(* Logix 5000 project; controller Sucrose_Main Emulate 5570 rev 20.12; software revision 20.01; part 15 of 30 *)
(* tags used below, declared in another part *)
   Alarm_ACK_Master_Timer : TIMER;
   DI_E22_0 : ALIAS FOR FLX_E22:0:I;   // Discrete Input EN2T_FLX 192.168.1.22
   DO_E22_2 : ALIAS FOR FLX_E22:2:O;   // Discrete Output EN2T_FLX 192.168.1.22
   DO_E22_3 : ALIAS FOR FLX_E22:3:O;   // Discrete Output EN2T_FLX 192.168.1.22
   DO_E22_4 : ALIAS FOR FLX_E22:4:O;   // Discrete Output EN2T_FLX 192.168.1.22
   FV140501_AOI : QSI_Flow_Valve;   // FV-14-05-01 PRE FILTER TRAIN 1 SUPPLY VALVE
   FV140502_AOI : QSI_Flow_Valve;   // FV-14-05-02 FINAL FILTER TRAIN 1 SUPPLY VALVE
   FV140503_AOI : QSI_Flow_Valve;   // FV-14-05-03 HOT WATER LOW POINT DRAIN VALVE
   FV140601_AOI : QSI_Flow_Valve;   // FV-14-06-01 PRE FILTER TRAIN 2 SUPPLY VALVE
   FV140602_AOI : QSI_Flow_Valve;   // FV-14-06-02 FINAL FILTER TRAIN 2 SUPPLY VALVE
   FV150501_AOI : QSI_Flow_Valve;   // FV-15-05-01 DIVERT TO SCRAP OR TO DRAIN VALVE
   FV230500_AOI : QSI_Flow_Valve;   // FV-23-05-00 SUCROSE LOW POINT DRAIN VALVE
   FV230601_AOI : QSI_Flow_Valve;   // FV-23-06-01-O PRE FILTER TRAIN 2 INLET VALVE OPEN
   FV230606_AOI : QSI_Flow_Valve;   // FV-23-06-06-O PRE FILTER TRAIN 2 OUTLET VALVE OPEN
   FV230608_AOI : QSI_Flow_Valve;   // FV-23-06-08-O FINAL FILTER TRAIN 2 INLET VALVE OPEN
   FV230613_AOI : QSI_Flow_Valve;   // FV-23-06-13-O FINAL FILTER TRAIN 2 OUTLET VALVE OPEN
   Sucrose_MM_Enable : BOOL;
   SucroseCIP_FILTRATION_REMOTE : CIP_REMOTE;
   SucroseFiltration : Area_Program;
(* FiltrationArea_EN2T_IO_Discrete_DO_E22_2, continued *)

ROUTINE _12_FV230601   (* ladder *)
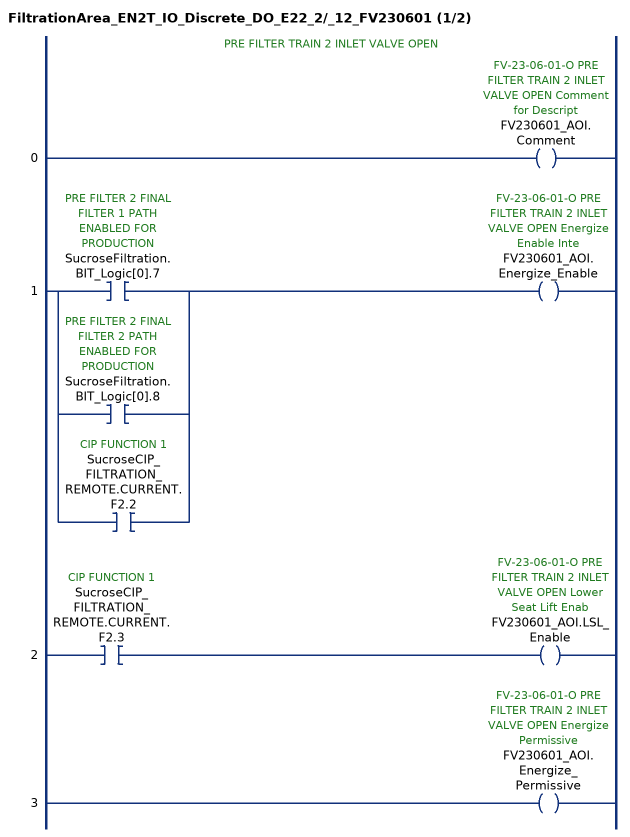
   // PRE FILTER TRAIN 2 INLET VALVE OPEN
   0: OTE(FV230601_AOI.Comment);
   1: [XIC(SucroseFiltration.BIT_Logic[0].7) ,XIC(SucroseFiltration.BIT_Logic[0].8) ,XIC(SucroseCIP_FILTRATION_REMOTE.CURRENT.F2.2) ]OTE(FV230601_AOI.Energize_Enable);
   2: XIC(SucroseCIP_FILTRATION_REMOTE.CURRENT.F2.3)OTE(FV230601_AOI.LSL_Enable);
   3: OTE(FV230601_AOI.Energize_Permissive);
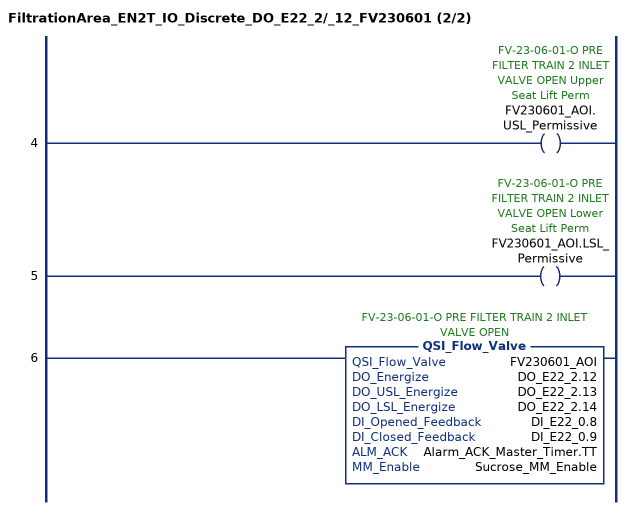
   4: OTE(FV230601_AOI.USL_Permissive);
   5: OTE(FV230601_AOI.LSL_Permissive);
   6: QSI_Flow_Valve(FV230601_AOI,DO_E22_2.12,DO_E22_2.13,DO_E22_2.14,DI_E22_0.8,DI_E22_0.9,Alarm_ACK_Master_Timer.TT,Sucrose_MM_Enable);
END_ROUTINE

ROUTINE MainRoutine   (* ladder *)
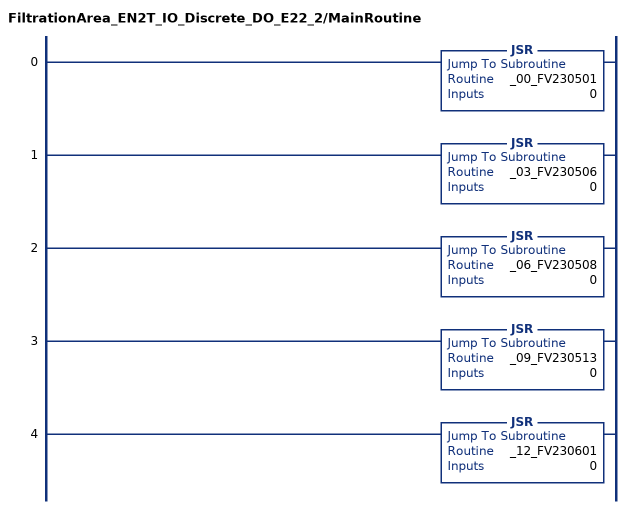
   0: JSR(_00_FV230501,0);
   1: JSR(_03_FV230506,0);
   2: JSR(_06_FV230508,0);
   3: JSR(_09_FV230513,0);
   4: JSR(_12_FV230601,0);
END_ROUTINE
END_PROGRAM

PROGRAM FiltrationArea_EN2T_IO_Discrete_DO_E22_3   (* main routine MainRoutine *)

ROUTINE _00_FV230606   (* ladder *)
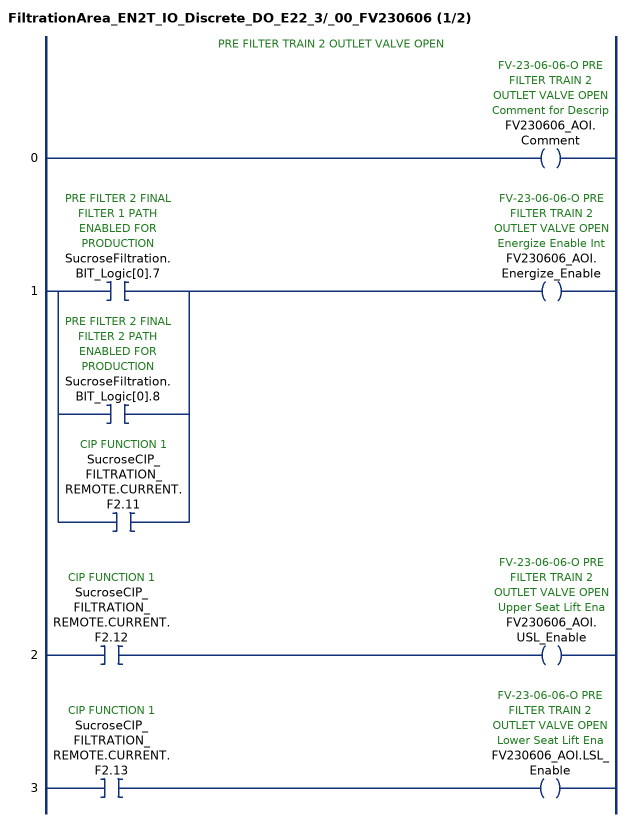
   // PRE FILTER TRAIN 2 OUTLET VALVE OPEN
   0: OTE(FV230606_AOI.Comment);
   1: [XIC(SucroseFiltration.BIT_Logic[0].7) ,XIC(SucroseFiltration.BIT_Logic[0].8) ,XIC(SucroseCIP_FILTRATION_REMOTE.CURRENT.F2.11) ]OTE(FV230606_AOI.Energize_Enable);
   2: XIC(SucroseCIP_FILTRATION_REMOTE.CURRENT.F2.12)OTE(FV230606_AOI.USL_Enable);
   3: XIC(SucroseCIP_FILTRATION_REMOTE.CURRENT.F2.13)OTE(FV230606_AOI.LSL_Enable);
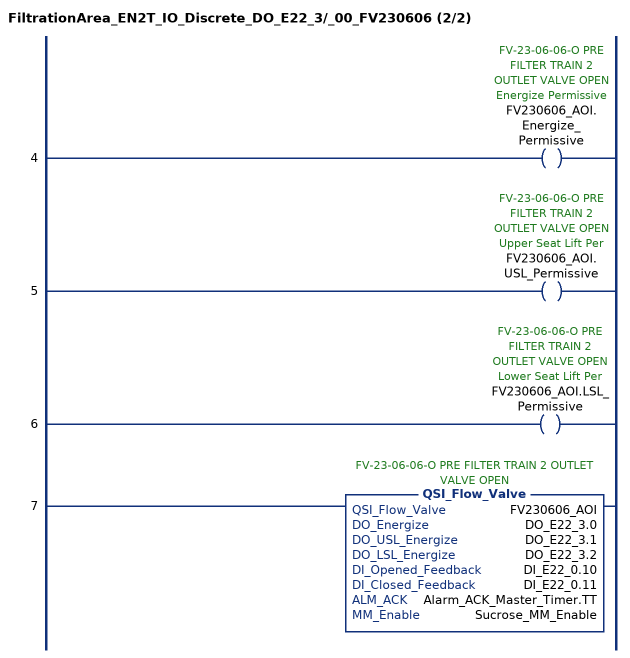
   4: OTE(FV230606_AOI.Energize_Permissive);
   5: OTE(FV230606_AOI.USL_Permissive);
   6: OTE(FV230606_AOI.LSL_Permissive);
   7: QSI_Flow_Valve(FV230606_AOI,DO_E22_3.0,DO_E22_3.1,DO_E22_3.2,DI_E22_0.10,DI_E22_0.11,Alarm_ACK_Master_Timer.TT,Sucrose_MM_Enable);
END_ROUTINE

ROUTINE _03_FV230608   (* ladder *)
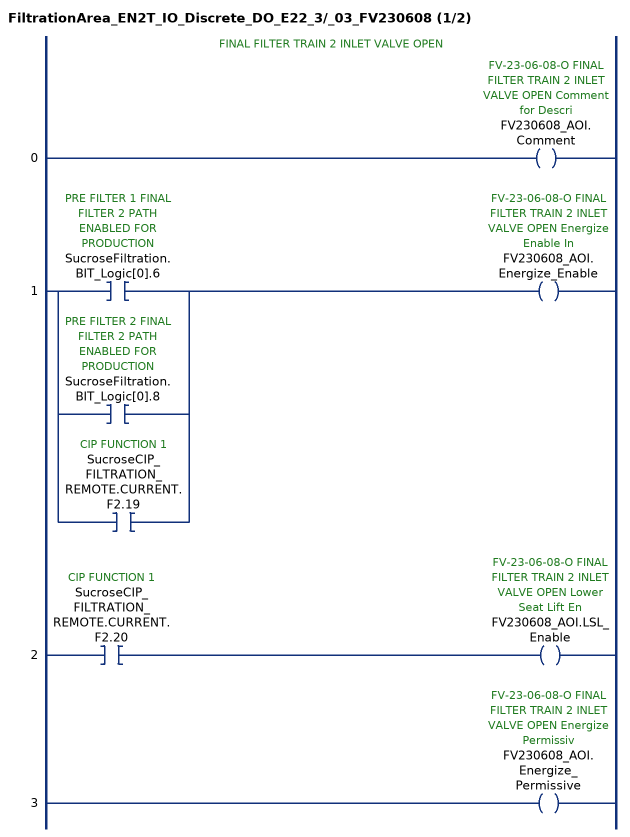
   // FINAL FILTER TRAIN 2 INLET VALVE OPEN
   0: OTE(FV230608_AOI.Comment);
   1: [XIC(SucroseFiltration.BIT_Logic[0].6) ,XIC(SucroseFiltration.BIT_Logic[0].8) ,XIC(SucroseCIP_FILTRATION_REMOTE.CURRENT.F2.19) ]OTE(FV230608_AOI.Energize_Enable);
   2: XIC(SucroseCIP_FILTRATION_REMOTE.CURRENT.F2.20)OTE(FV230608_AOI.LSL_Enable);
   3: OTE(FV230608_AOI.Energize_Permissive);
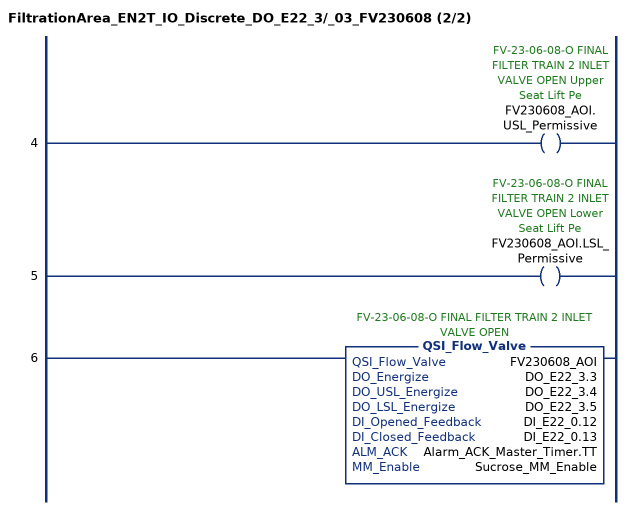
   4: OTE(FV230608_AOI.USL_Permissive);
   5: OTE(FV230608_AOI.LSL_Permissive);
   6: QSI_Flow_Valve(FV230608_AOI,DO_E22_3.3,DO_E22_3.4,DO_E22_3.5,DI_E22_0.12,DI_E22_0.13,Alarm_ACK_Master_Timer.TT,Sucrose_MM_Enable);
END_ROUTINE

ROUTINE _06_FV230613   (* ladder *)
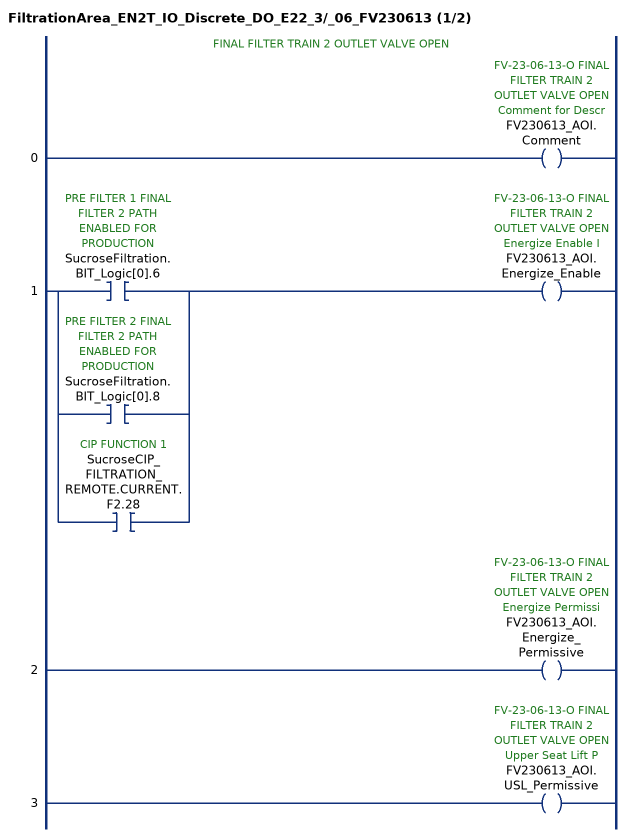
   // FINAL FILTER TRAIN 2 OUTLET VALVE OPEN
   0: OTE(FV230613_AOI.Comment);
   1: [XIC(SucroseFiltration.BIT_Logic[0].6) ,XIC(SucroseFiltration.BIT_Logic[0].8) ,XIC(SucroseCIP_FILTRATION_REMOTE.CURRENT.F2.28) ]OTE(FV230613_AOI.Energize_Enable);
   2: OTE(FV230613_AOI.Energize_Permissive);
   3: OTE(FV230613_AOI.USL_Permissive);
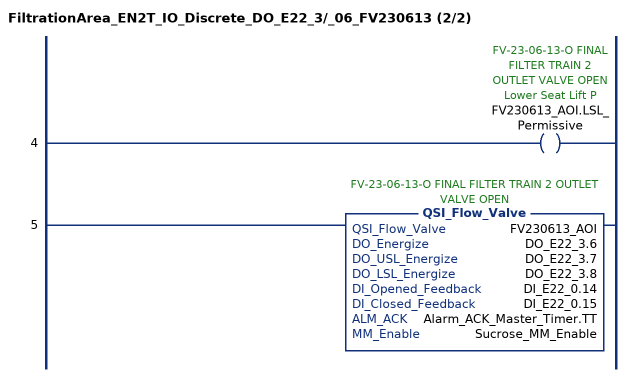
   4: OTE(FV230613_AOI.LSL_Permissive);
   5: QSI_Flow_Valve(FV230613_AOI,DO_E22_3.6,DO_E22_3.7,DO_E22_3.8,DI_E22_0.14,DI_E22_0.15,Alarm_ACK_Master_Timer.TT,Sucrose_MM_Enable);
END_ROUTINE

ROUTINE MainRoutine   (* ladder *)
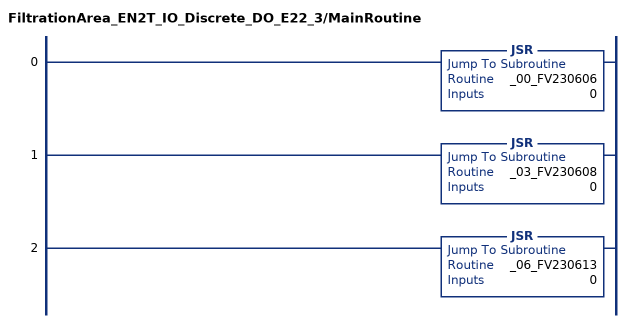
   0: JSR(_00_FV230606,0);
   1: JSR(_03_FV230608,0);
   2: JSR(_06_FV230613,0);
END_ROUTINE
END_PROGRAM

PROGRAM FiltrationArea_EN2T_IO_Discrete_DO_E22_4   (* main routine MainRoutine *)

ROUTINE _00_FV140501   (* ladder *)
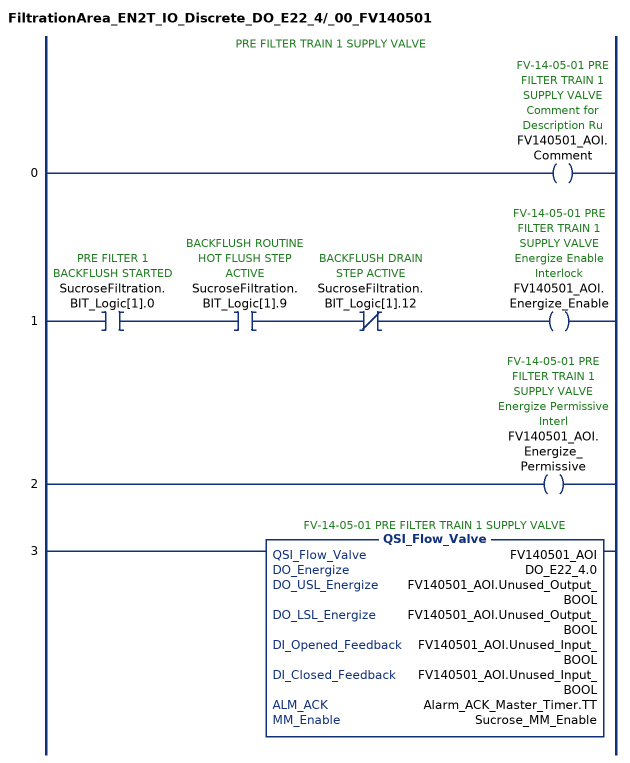
   // PRE FILTER TRAIN 1 SUPPLY VALVE
   0: OTE(FV140501_AOI.Comment);
   1: XIC(SucroseFiltration.BIT_Logic[1].0)XIC(SucroseFiltration.BIT_Logic[1].9)XIO(SucroseFiltration.BIT_Logic[1].12)OTE(FV140501_AOI.Energize_Enable);
   2: OTE(FV140501_AOI.Energize_Permissive);
   3: QSI_Flow_Valve(FV140501_AOI,DO_E22_4.0,FV140501_AOI.Unused_Output_BOOL,FV140501_AOI.Unused_Output_BOOL,FV140501_AOI.Unused_Input_BOOL,FV140501_AOI.Unused_Input_BOOL,Alarm_ACK_Master_Timer.TT,Sucrose_MM_Enable);
END_ROUTINE

ROUTINE _01_FV140502   (* ladder *)
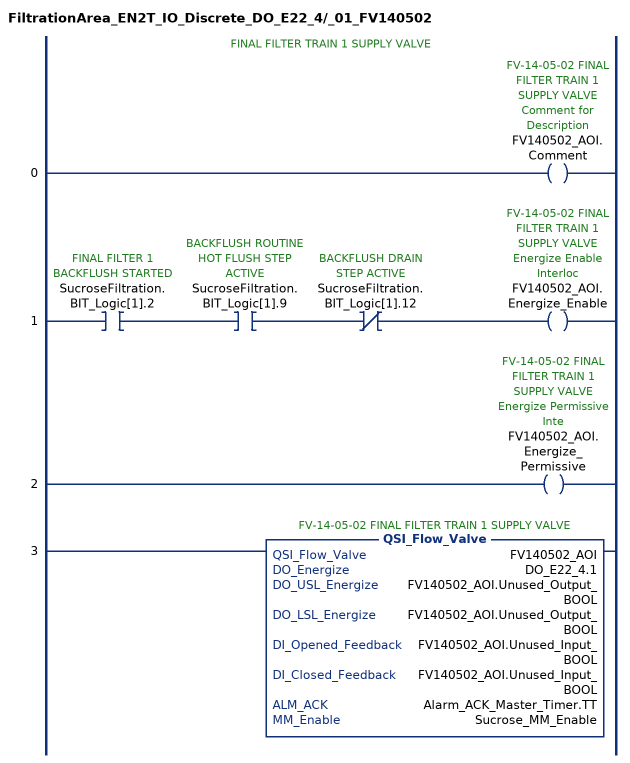
   // FINAL FILTER TRAIN 1 SUPPLY VALVE
   0: OTE(FV140502_AOI.Comment);
   1: XIC(SucroseFiltration.BIT_Logic[1].2)XIC(SucroseFiltration.BIT_Logic[1].9)XIO(SucroseFiltration.BIT_Logic[1].12)OTE(FV140502_AOI.Energize_Enable);
   2: OTE(FV140502_AOI.Energize_Permissive);
   3: QSI_Flow_Valve(FV140502_AOI,DO_E22_4.1,FV140502_AOI.Unused_Output_BOOL,FV140502_AOI.Unused_Output_BOOL,FV140502_AOI.Unused_Input_BOOL,FV140502_AOI.Unused_Input_BOOL,Alarm_ACK_Master_Timer.TT,Sucrose_MM_Enable);
END_ROUTINE

ROUTINE _02_FV140503   (* ladder *)
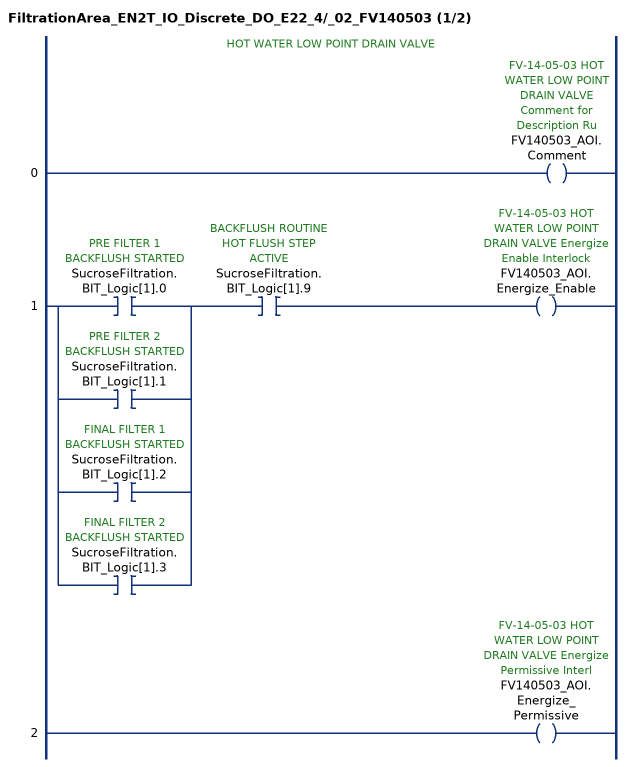
   // HOT WATER LOW POINT DRAIN VALVE
   0: OTE(FV140503_AOI.Comment);
   1: [XIC(SucroseFiltration.BIT_Logic[1].0) ,XIC(SucroseFiltration.BIT_Logic[1].1) ,XIC(SucroseFiltration.BIT_Logic[1].2) ,XIC(SucroseFiltration.BIT_Logic[1].3) ]XIC(SucroseFiltration.BIT_Logic[1].9)OTE(FV140503_AOI.Energize_Enable);
   2: OTE(FV140503_AOI.Energize_Permissive);
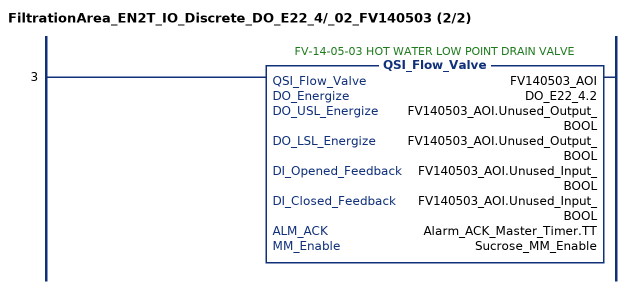
   3: QSI_Flow_Valve(FV140503_AOI,DO_E22_4.2,FV140503_AOI.Unused_Output_BOOL,FV140503_AOI.Unused_Output_BOOL,FV140503_AOI.Unused_Input_BOOL,FV140503_AOI.Unused_Input_BOOL,Alarm_ACK_Master_Timer.TT,Sucrose_MM_Enable);
END_ROUTINE

ROUTINE _03_FV140601   (* ladder *)
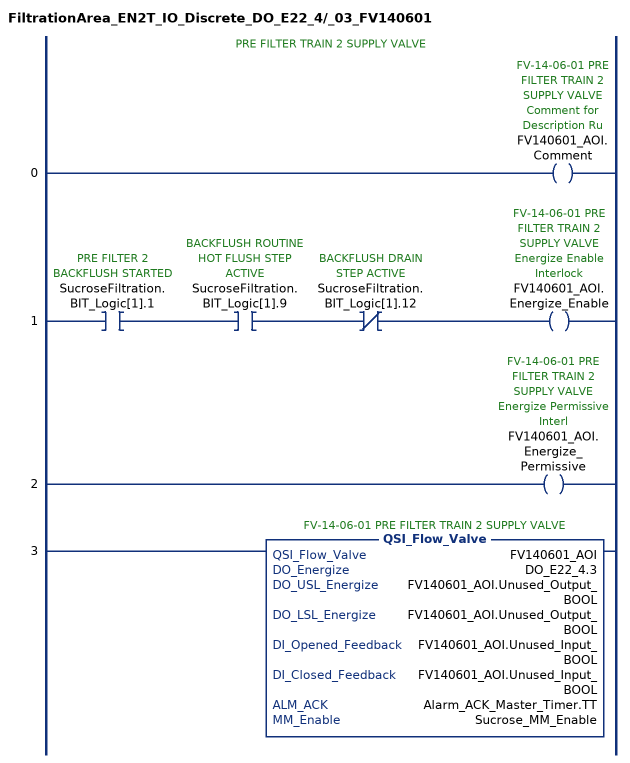
   // PRE FILTER TRAIN 2 SUPPLY VALVE
   0: OTE(FV140601_AOI.Comment);
   1: XIC(SucroseFiltration.BIT_Logic[1].1)XIC(SucroseFiltration.BIT_Logic[1].9)XIO(SucroseFiltration.BIT_Logic[1].12)OTE(FV140601_AOI.Energize_Enable);
   2: OTE(FV140601_AOI.Energize_Permissive);
   3: QSI_Flow_Valve(FV140601_AOI,DO_E22_4.3,FV140601_AOI.Unused_Output_BOOL,FV140601_AOI.Unused_Output_BOOL,FV140601_AOI.Unused_Input_BOOL,FV140601_AOI.Unused_Input_BOOL,Alarm_ACK_Master_Timer.TT,Sucrose_MM_Enable);
END_ROUTINE

ROUTINE _04_FV140602   (* ladder *)
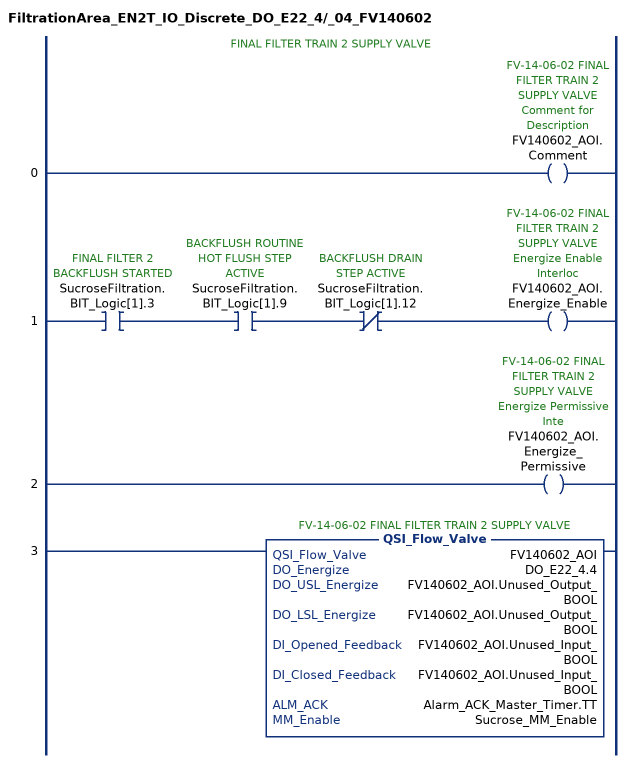
   // FINAL FILTER TRAIN 2 SUPPLY VALVE
   0: OTE(FV140602_AOI.Comment);
   1: XIC(SucroseFiltration.BIT_Logic[1].3)XIC(SucroseFiltration.BIT_Logic[1].9)XIO(SucroseFiltration.BIT_Logic[1].12)OTE(FV140602_AOI.Energize_Enable);
   2: OTE(FV140602_AOI.Energize_Permissive);
   3: QSI_Flow_Valve(FV140602_AOI,DO_E22_4.4,FV140602_AOI.Unused_Output_BOOL,FV140602_AOI.Unused_Output_BOOL,FV140602_AOI.Unused_Input_BOOL,FV140602_AOI.Unused_Input_BOOL,Alarm_ACK_Master_Timer.TT,Sucrose_MM_Enable);
END_ROUTINE

ROUTINE _05_FV150501   (* ladder *)
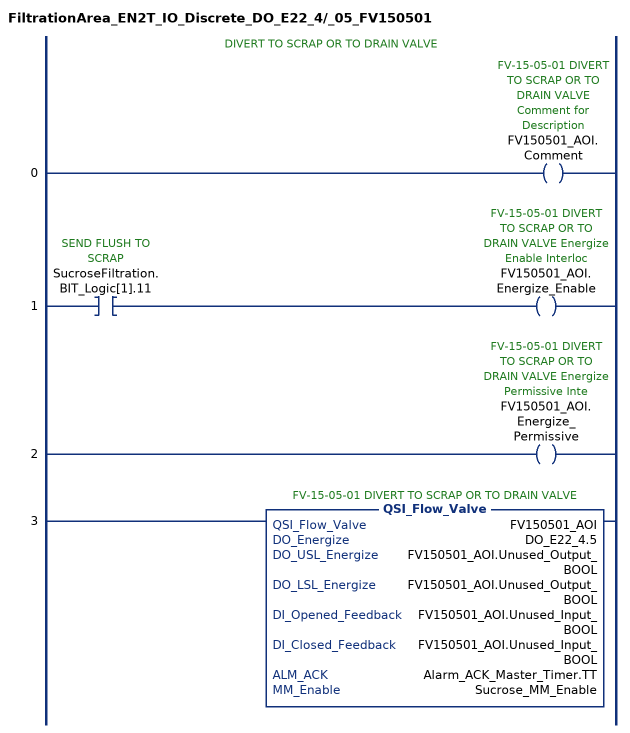
   // DIVERT TO SCRAP OR TO DRAIN VALVE
   0: OTE(FV150501_AOI.Comment);
   1: XIC(SucroseFiltration.BIT_Logic[1].11)OTE(FV150501_AOI.Energize_Enable);
   2: OTE(FV150501_AOI.Energize_Permissive);
   3: QSI_Flow_Valve(FV150501_AOI,DO_E22_4.5,FV150501_AOI.Unused_Output_BOOL,FV150501_AOI.Unused_Output_BOOL,FV150501_AOI.Unused_Input_BOOL,FV150501_AOI.Unused_Input_BOOL,Alarm_ACK_Master_Timer.TT,Sucrose_MM_Enable);
END_ROUTINE

ROUTINE _06_FV230500   (* ladder *)
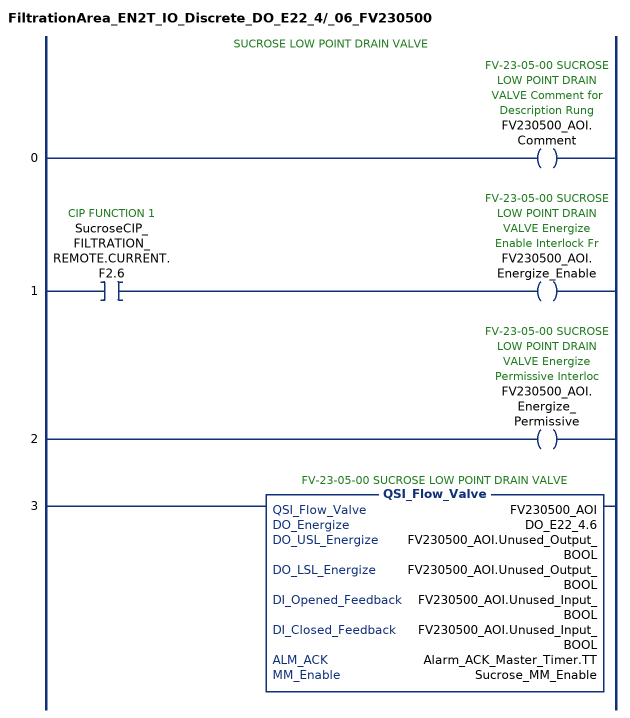
   // SUCROSE LOW POINT DRAIN VALVE
   0: OTE(FV230500_AOI.Comment);
   1: XIC(SucroseCIP_FILTRATION_REMOTE.CURRENT.F2.6)OTE(FV230500_AOI.Energize_Enable);
   2: OTE(FV230500_AOI.Energize_Permissive);
   3: QSI_Flow_Valve(FV230500_AOI,DO_E22_4.6,FV230500_AOI.Unused_Output_BOOL,FV230500_AOI.Unused_Output_BOOL,FV230500_AOI.Unused_Input_BOOL,FV230500_AOI.Unused_Input_BOOL,Alarm_ACK_Master_Timer.TT,Sucrose_MM_Enable);
END_ROUTINE
